// TIA Portal V19 export
FUNCTION "JB_CALL" : Void   // FC127, LAD
TITLE = JUNCTION BENCH WELDER CALL
// stored: SetENOAutomatically false
BEGIN

REGION Network 1: Data In - Welder speed potentiometer
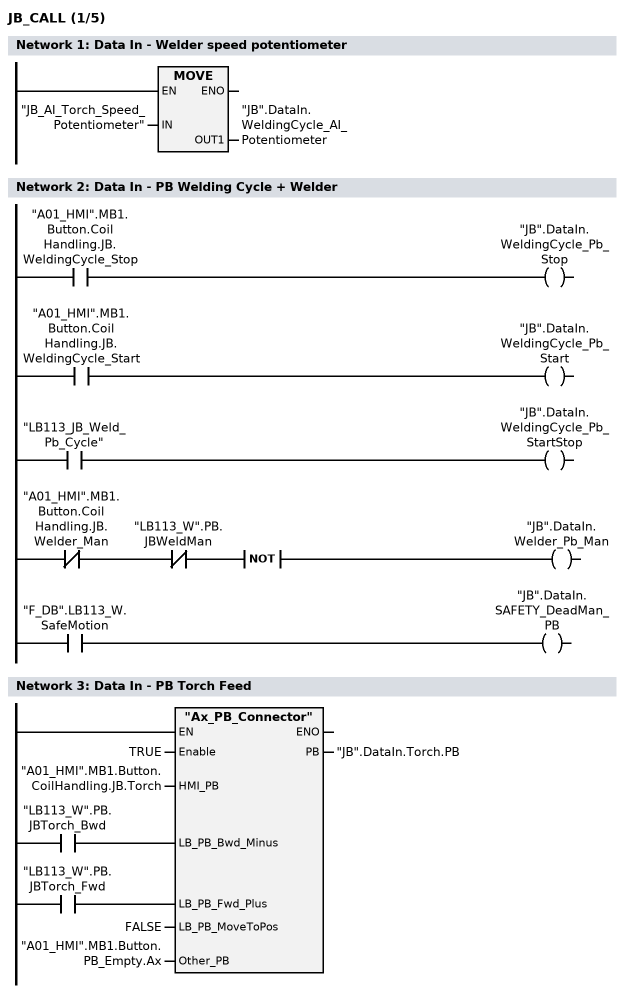
   RUNG wire#powerrail
      Move(in := "JB_AI_Torch_Speed_Potentiometer", out1 => "JB".DataIn.WeldingCycle_AI_Potentiometer)
   END_RUNG
   // the same network as SCL:
   "JB".DataIn.WeldingCycle_AI_Potentiometer := "JB_AI_Torch_Speed_Potentiometer";
END_REGION

REGION Network 2: Data In - PB Welding Cycle + Welder
   RUNG wire#powerrail
      Contact( "A01_HMI".MB1.Button.CoilHandling.JB.WeldingCycle_Stop )
      Coil( "JB".DataIn.WeldingCycle_Pb_Stop )
   END_RUNG
   RUNG wire#powerrail
      Contact( "A01_HMI".MB1.Button.CoilHandling.JB.WeldingCycle_Start )
      Coil( "JB".DataIn.WeldingCycle_Pb_Start )
   END_RUNG
   RUNG wire#powerrail
      Contact( "LB113_JB_Weld_Pb_Cycle" )
      Coil( "JB".DataIn.WeldingCycle_Pb_StartStop )
   END_RUNG
   RUNG wire#powerrail
      I_Contact( "A01_HMI".MB1.Button.CoilHandling.JB.Welder_Man )
      I_Contact( "LB113_W".PB.JBWeldMan )
      Not()
      Coil( "JB".DataIn.Welder_Pb_Man )
   END_RUNG
   RUNG wire#powerrail
      Contact( "F_DB".LB113_W.SafeMotion )
      Coil( "JB".DataIn.SAFETY_DeadMan_PB )
   END_RUNG
   // the same network as SCL:
   "JB".DataIn.WeldingCycle_Pb_Stop := "A01_HMI".MB1.Button.CoilHandling.JB.WeldingCycle_Stop;
   "JB".DataIn.WeldingCycle_Pb_Start := "A01_HMI".MB1.Button.CoilHandling.JB.WeldingCycle_Start;
   "JB".DataIn.WeldingCycle_Pb_StartStop := "LB113_JB_Weld_Pb_Cycle";
   "JB".DataIn.Welder_Pb_Man := NOT (NOT "A01_HMI".MB1.Button.CoilHandling.JB.Welder_Man AND NOT "LB113_W".PB.JBWeldMan);
   "JB".DataIn.SAFETY_DeadMan_PB := "F_DB".LB113_W.SafeMotion;
END_REGION

REGION Network 3: Data In - PB Torch Feed
   RUNG wire#powerrail
      "Ax_PB_Connector"(LB_PB_Bwd_Minus := wire#w1, LB_PB_Fwd_Plus := wire#w2, Enable := TRUE, HMI_PB := "A01_HMI".MB1.Button.CoilHandling.JB.Torch, LB_PB_MoveToPos := FALSE, Other_PB := "A01_HMI".MB1.Button.PB_Empty.Ax, PB => "JB".DataIn.Torch.PB)
   END_RUNG
   RUNG wire#powerrail
      Contact( "LB113_W".PB.JBTorch_Bwd )
   END_RUNG wire#w1
   RUNG wire#powerrail
      Contact( "LB113_W".PB.JBTorch_Fwd )
   END_RUNG wire#w2
   // the same network as SCL:
   "Ax_PB_Connector"(Enable := TRUE,
                     HMI_PB := "A01_HMI".MB1.Button.CoilHandling.JB.Torch,
                     LB_PB_Bwd_Minus := "LB113_W".PB.JBTorch_Bwd,
                     LB_PB_Fwd_Plus := "LB113_W".PB.JBTorch_Fwd,
                     LB_PB_MoveToPos := FALSE,
                     Other_PB := "A01_HMI".MB1.Button.PB_Empty.Ax,
                     PB => "JB".DataIn.Torch.PB);
END_REGION

REGION Network 4: Data In - PB Clamps
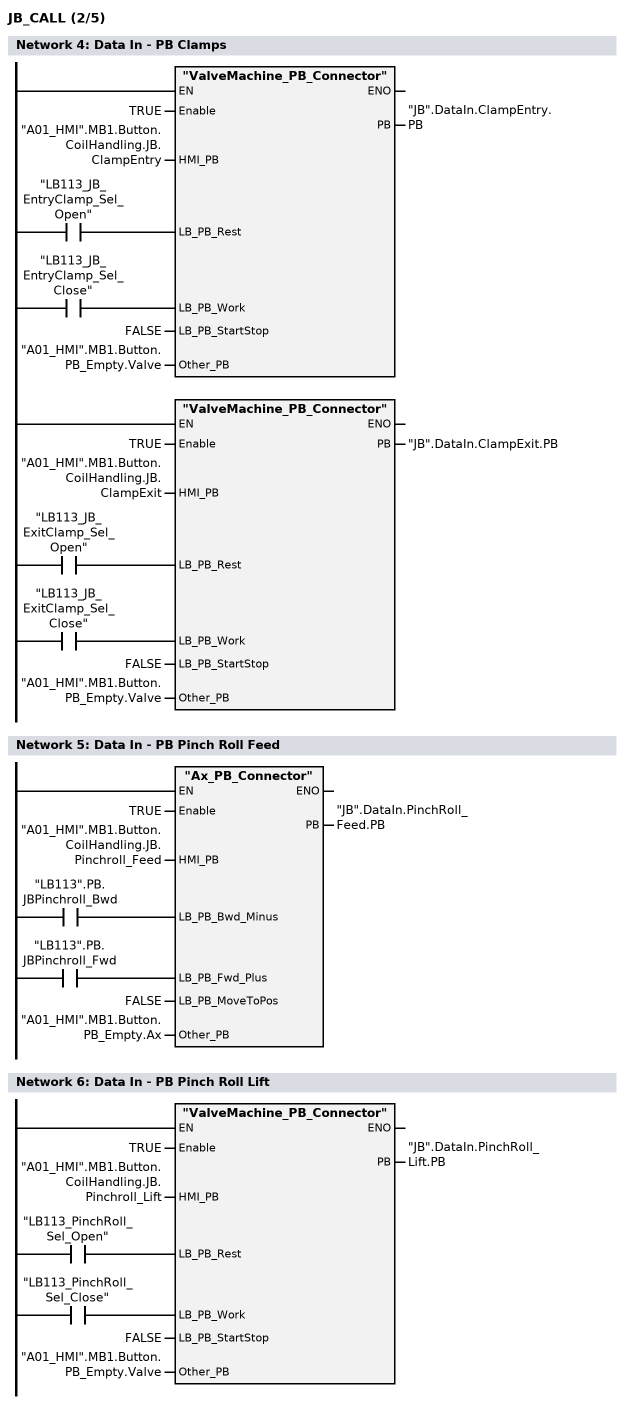
   RUNG wire#powerrail
      "ValveMachine_PB_Connector"(LB_PB_Rest := wire#w1, LB_PB_Work := wire#w2, Enable := TRUE, HMI_PB := "A01_HMI".MB1.Button.CoilHandling.JB.ClampEntry, LB_PB_StartStop := FALSE, Other_PB := "A01_HMI".MB1.Button.PB_Empty.Valve, PB => "JB".DataIn.ClampEntry.PB)
   END_RUNG
   RUNG wire#powerrail
      Contact( "LB113_JB_EntryClamp_Sel_Open" )
   END_RUNG wire#w1
   RUNG wire#powerrail
      Contact( "LB113_JB_EntryClamp_Sel_Close" )
   END_RUNG wire#w2
   RUNG wire#powerrail
      "ValveMachine_PB_Connector"(LB_PB_Rest := wire#w3, LB_PB_Work := wire#w4, Enable := TRUE, HMI_PB := "A01_HMI".MB1.Button.CoilHandling.JB.ClampExit, LB_PB_StartStop := FALSE, Other_PB := "A01_HMI".MB1.Button.PB_Empty.Valve, PB => "JB".DataIn.ClampExit.PB)
   END_RUNG
   RUNG wire#powerrail
      Contact( "LB113_JB_ExitClamp_Sel_Open" )
   END_RUNG wire#w3
   RUNG wire#powerrail
      Contact( "LB113_JB_ExitClamp_Sel_Close" )
   END_RUNG wire#w4
   // the same network as SCL:
   "ValveMachine_PB_Connector"(Enable := TRUE,
                           HMI_PB := "A01_HMI".MB1.Button.CoilHandling.JB.ClampEntry,
                           LB_PB_Rest := "LB113_JB_EntryClamp_Sel_Open",
                           LB_PB_Work := "LB113_JB_EntryClamp_Sel_Close",
                           LB_PB_StartStop := FALSE,
                           Other_PB := "A01_HMI".MB1.Button.PB_Empty.Valve,
                           PB => "JB".DataIn.ClampEntry.PB);
   "ValveMachine_PB_Connector"(Enable := TRUE,
                           HMI_PB := "A01_HMI".MB1.Button.CoilHandling.JB.ClampExit,
                           LB_PB_Rest := "LB113_JB_ExitClamp_Sel_Open",
                           LB_PB_Work := "LB113_JB_ExitClamp_Sel_Close",
                           LB_PB_StartStop := FALSE,
                           Other_PB := "A01_HMI".MB1.Button.PB_Empty.Valve,
                           PB => "JB".DataIn.ClampExit.PB);
END_REGION

REGION Network 5: Data In - PB Pinch Roll Feed
   RUNG wire#powerrail
      "Ax_PB_Connector"(LB_PB_Bwd_Minus := wire#w1, LB_PB_Fwd_Plus := wire#w2, Enable := TRUE, HMI_PB := "A01_HMI".MB1.Button.CoilHandling.JB.Pinchroll_Feed, LB_PB_MoveToPos := FALSE, Other_PB := "A01_HMI".MB1.Button.PB_Empty.Ax, PB => "JB".DataIn.PinchRoll_Feed.PB)
   END_RUNG
   RUNG wire#powerrail
      Contact( "LB113".PB.JBPinchroll_Bwd )
   END_RUNG wire#w1
   RUNG wire#powerrail
      Contact( "LB113".PB.JBPinchroll_Fwd )
   END_RUNG wire#w2
   // the same network as SCL:
   "Ax_PB_Connector"(Enable := TRUE,
                     HMI_PB := "A01_HMI".MB1.Button.CoilHandling.JB.Pinchroll_Feed,
                     LB_PB_Bwd_Minus := "LB113".PB.JBPinchroll_Bwd,
                     LB_PB_Fwd_Plus := "LB113".PB.JBPinchroll_Fwd,
                     LB_PB_MoveToPos := FALSE,
                     Other_PB := "A01_HMI".MB1.Button.PB_Empty.Ax,
                     PB => "JB".DataIn.PinchRoll_Feed.PB);
END_REGION

REGION Network 6: Data In - PB Pinch Roll Lift
   RUNG wire#powerrail
      "ValveMachine_PB_Connector"(LB_PB_Rest := wire#w1, LB_PB_Work := wire#w2, Enable := TRUE, HMI_PB := "A01_HMI".MB1.Button.CoilHandling.JB.Pinchroll_Lift, LB_PB_StartStop := FALSE, Other_PB := "A01_HMI".MB1.Button.PB_Empty.Valve, PB => "JB".DataIn.PinchRoll_Lift.PB)
   END_RUNG
   RUNG wire#powerrail
      Contact( "LB113_PinchRoll_Sel_Open" )
   END_RUNG wire#w1
   RUNG wire#powerrail
      Contact( "LB113_PinchRoll_Sel_Close" )
   END_RUNG wire#w2
   // the same network as SCL:
   "ValveMachine_PB_Connector"(Enable := TRUE,
                           HMI_PB := "A01_HMI".MB1.Button.CoilHandling.JB.Pinchroll_Lift,
                           LB_PB_Rest := "LB113_PinchRoll_Sel_Open",
                           LB_PB_Work := "LB113_PinchRoll_Sel_Close",
                           LB_PB_StartStop := FALSE,
                           Other_PB := "A01_HMI".MB1.Button.PB_Empty.Valve,
                           PB => "JB".DataIn.PinchRoll_Lift.PB);
END_REGION

REGION Network 7: Data In - PB Cut Head
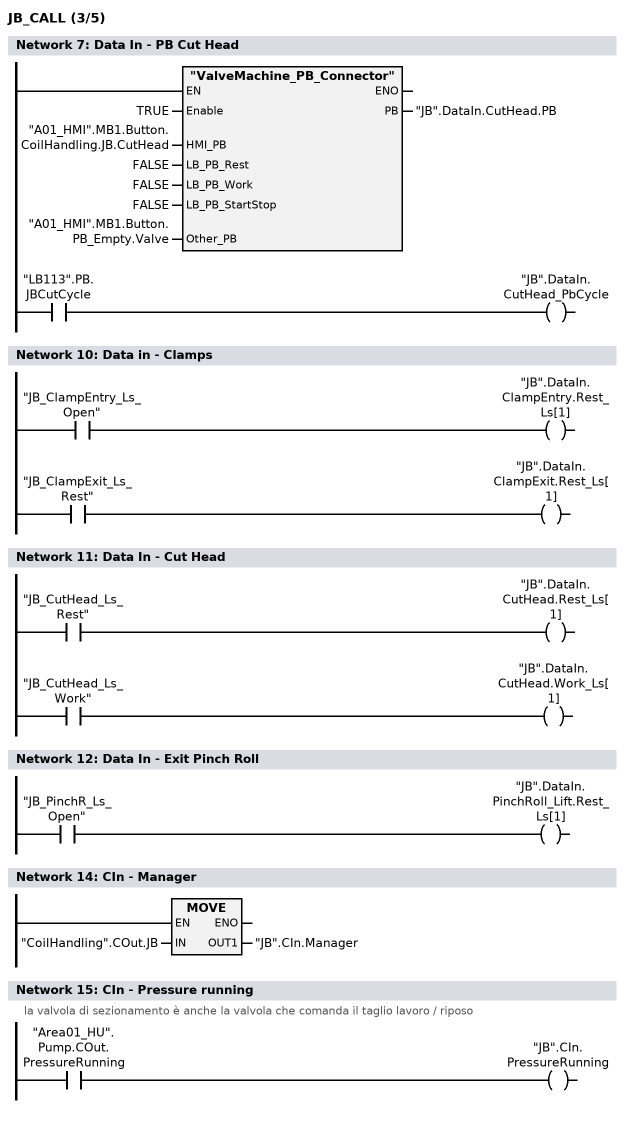
   RUNG wire#powerrail
      "ValveMachine_PB_Connector"(Enable := TRUE, HMI_PB := "A01_HMI".MB1.Button.CoilHandling.JB.CutHead, LB_PB_Rest := FALSE, LB_PB_Work := FALSE, LB_PB_StartStop := FALSE, Other_PB := "A01_HMI".MB1.Button.PB_Empty.Valve, PB => "JB".DataIn.CutHead.PB)
   END_RUNG
   RUNG wire#powerrail
      Contact( "LB113".PB.JBCutCycle )
      Coil( "JB".DataIn.CutHead_PbCycle )
   END_RUNG
   // the same network as SCL:
   "ValveMachine_PB_Connector"(Enable := TRUE,
                           HMI_PB := "A01_HMI".MB1.Button.CoilHandling.JB.CutHead,
                           LB_PB_Rest := FALSE,
                           LB_PB_Work := FALSE,
                           LB_PB_StartStop := FALSE,
                           Other_PB := "A01_HMI".MB1.Button.PB_Empty.Valve,
                           PB => "JB".DataIn.CutHead.PB);
   "JB".DataIn.CutHead_PbCycle := "LB113".PB.JBCutCycle;
END_REGION

REGION Network 8: >
END_REGION

REGION Network 9: >
END_REGION

REGION Network 10: Data in - Clamps
   RUNG wire#powerrail
      Contact( "JB_ClampEntry_Ls_Open" )
      Coil( "JB".DataIn.ClampEntry.Rest_Ls[1] )
   END_RUNG
   RUNG wire#powerrail
      Contact( "JB_ClampExit_Ls_Rest" )
      Coil( "JB".DataIn.ClampExit.Rest_Ls[1] )
   END_RUNG
   // the same network as SCL:
   "JB".DataIn.ClampEntry.Rest_Ls[1] := "JB_ClampEntry_Ls_Open";
   "JB".DataIn.ClampExit.Rest_Ls[1] := "JB_ClampExit_Ls_Rest";
END_REGION

REGION Network 11: Data In - Cut Head
   RUNG wire#powerrail
      Contact( "JB_CutHead_Ls_Rest" )
      Coil( "JB".DataIn.CutHead.Rest_Ls[1] )
   END_RUNG
   RUNG wire#powerrail
      Contact( "JB_CutHead_Ls_Work" )
      Coil( "JB".DataIn.CutHead.Work_Ls[1] )
   END_RUNG
   // the same network as SCL:
   "JB".DataIn.CutHead.Rest_Ls[1] := "JB_CutHead_Ls_Rest";
   "JB".DataIn.CutHead.Work_Ls[1] := "JB_CutHead_Ls_Work";
END_REGION

REGION Network 12: Data In - Exit Pinch Roll
   RUNG wire#powerrail
      Contact( "JB_PinchR_Ls_Open" )
      Coil( "JB".DataIn.PinchRoll_Lift.Rest_Ls[1] )
   END_RUNG
   // the same network as SCL:
   "JB".DataIn.PinchRoll_Lift.Rest_Ls[1] := "JB_PinchR_Ls_Open";
END_REGION

REGION Network 13: >
END_REGION

REGION Network 14: CIn - Manager
   RUNG wire#powerrail
      Move(in := "CoilHandling".COut.JB, out1 => "JB".CIn.Manager)
   END_RUNG
   // the same network as SCL:
   "JB".CIn.Manager := "CoilHandling".COut.JB;
END_REGION

REGION Network 15: CIn - Pressure running
   // la valvola di sezionamento è anche la valvola che comanda il taglio lavoro / riposo
   RUNG wire#powerrail
      Contact( "Area01_HU".Pump.COut.PressureRunning )
      Coil( "JB".CIn.PressureRunning )
   END_RUNG
   // the same network as SCL:
   "JB".CIn.PressureRunning := "Area01_HU".Pump.COut.PressureRunning;
END_REGION

REGION Network 16: >
END_REGION

REGION Network 17 (SCL): DSI
   "JB".DSI.Torch := "F_DB".DSI_S120_JB_Torch;

   "JB".DSI.PinchRoll_Feed := "F_DB".DSI_S120_JB_PinchRoll;

   "JB".DSI.ClampEntry :=
   "JB".DSI.ClampExit :=
   "JB".DSI.PinchRoll_Lift := "F_DB".DSI_V_Air_Gen;


   // Cut Head
   IF "JB".CutHead.COut.Rest_CheckNext THEN

       "JB".DSI.CutHead.SafeStop := "F_DB".DSI_V_JB_Cut_Rest.SafeStop;
       "JB".DSI.CutHead.PowerEnable := "F_DB".DSI_V_JB_Cut_Rest.PowerEnable;
       "JB".DSI.CutHead.DevicesInSafeState := "F_DB".DSI_V_JB_Cut_Rest.DevicesInSafeState;

   ELSIF "JB".CutHead.COut.Work_CheckNext THEN

       "JB".DSI.CutHead.SafeStop := "F_DB".DSI_V_JB_Cut_Work.SafeStop;
       "JB".DSI.CutHead.PowerEnable := "F_DB".DSI_V_JB_Cut_Work.PowerEnable;
       "JB".DSI.CutHead.DevicesInSafeState := "F_DB".DSI_V_JB_Cut_Work.DevicesInSafeState;

   ELSE
       "JB".DSI.CutHead.SafeStop := TRUE;
       "JB".DSI.CutHead.PowerEnable := FALSE;
       "JB".DSI.CutHead.DevicesInSafeState := TRUE;
   END_IF;
END_REGION

REGION Network 18 (SCL): Drive
   "JB".Drive.Torch.Infeed_ON := "Areas_ITF".AG.Infeed_Running;
   "JB".Drive.Torch.AccessPoint := "HW_Const_Values".CU1_PN_890A1_1_ModuleAccessPoint;
   "JB".Drive.Torch.AxisID := "CU1_ID_7_890A1_1_890M1";
   "JB".Drive.Torch.TokenChain := "TOKENCHAIN_CU1";

   "JB".Drive.Picnhroll_Feed.Infeed_ON := "Areas_ITF".AG.Infeed_Running;
   "JB".Drive.Picnhroll_Feed.AccessPoint := "CU1~PN~890A1_2_ModuleAccessPoint";
   "JB".Drive.Picnhroll_Feed.AxisID := "CU1_ID_8_890A1_2_900M1";
   "JB".Drive.Picnhroll_Feed.TokenChain := "TOKENCHAIN_CU1";
END_REGION

REGION Network 19 (SCL): HW ID
   "JB".HWID.Torch_TEL1 := "HW_Const_Values".CU1_PN_890A1_1_Standard_telegram_1;
   "JB".HWID.Pinchroll_Feed_TEL1 := "HW_Const_Values".CU1_PN_890A1_2_Standard_telegram_1;
   "JB".HWID.TorchEnc_IO := "HW_Const_Values".HW_894P1_Telegram_81_DI_DO;
END_REGION

REGION Network 20: >
END_REGION

REGION Network 21: Machine Manager
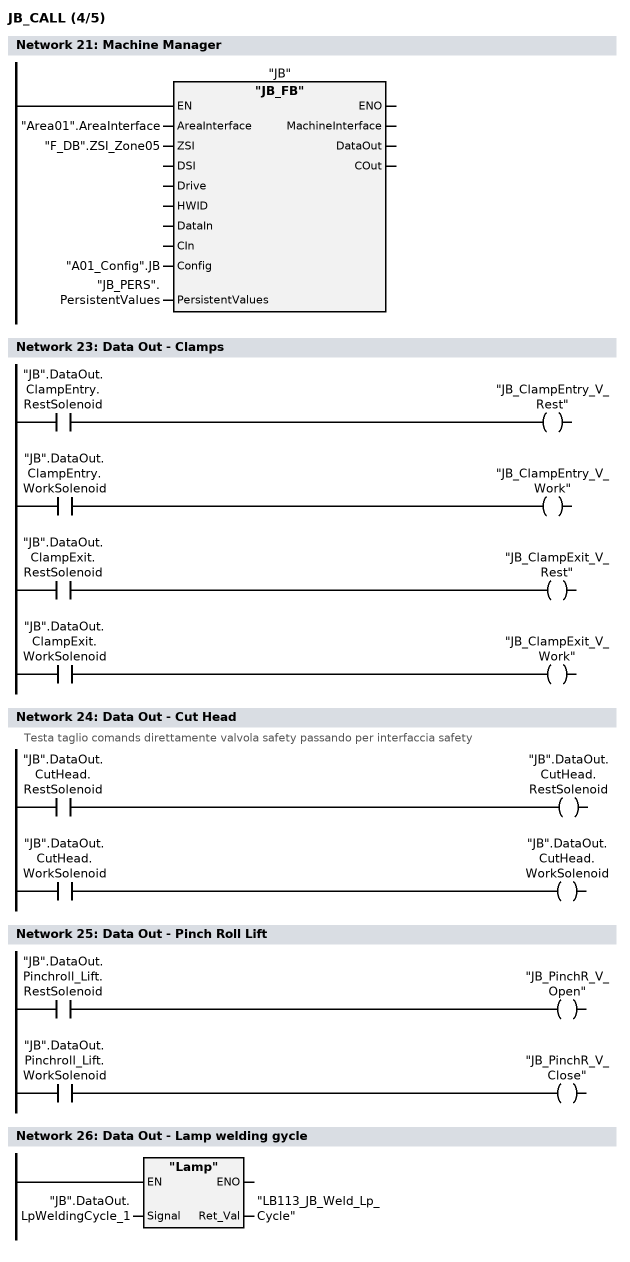
   RUNG wire#powerrail
      "JB"(AreaInterface := "Area01".AreaInterface, ZSI := "F_DB".ZSI_Zone05, DSI :=, Drive :=, HWID :=, DataIn :=, CIn :=, Config := "A01_Config".JB, PersistentValues := "JB_PERS".PersistentValues, MachineInterface =>, DataOut =>, COut =>)
   END_RUNG
   // the same network as SCL:
   "JB"(AreaInterface := "Area01".AreaInterface,   // "JB_FB"
        ZSI := "F_DB".ZSI_Zone05,
        Config := "A01_Config".JB,
        PersistentValues := "JB_PERS".PersistentValues);
END_REGION

REGION Network 22: >
END_REGION

REGION Network 23: Data Out - Clamps
   RUNG wire#powerrail
      Contact( "JB".DataOut.ClampEntry.RestSolenoid )
      Coil( "JB_ClampEntry_V_Rest" )
   END_RUNG
   RUNG wire#powerrail
      Contact( "JB".DataOut.ClampEntry.WorkSolenoid )
      Coil( "JB_ClampEntry_V_Work" )
   END_RUNG
   RUNG wire#powerrail
      Contact( "JB".DataOut.ClampExit.RestSolenoid )
      Coil( "JB_ClampExit_V_Rest" )
   END_RUNG
   RUNG wire#powerrail
      Contact( "JB".DataOut.ClampExit.WorkSolenoid )
      Coil( "JB_ClampExit_V_Work" )
   END_RUNG
   // the same network as SCL:
   "JB_ClampEntry_V_Rest" := "JB".DataOut.ClampEntry.RestSolenoid;
   "JB_ClampEntry_V_Work" := "JB".DataOut.ClampEntry.WorkSolenoid;
   "JB_ClampExit_V_Rest" := "JB".DataOut.ClampExit.RestSolenoid;
   "JB_ClampExit_V_Work" := "JB".DataOut.ClampExit.WorkSolenoid;
END_REGION

REGION Network 24: Data Out - Cut Head
   // Testa taglio comands direttamente valvola safety passando per interfaccia safety
   RUNG wire#powerrail
      Contact( "JB".DataOut.CutHead.RestSolenoid )
      Coil( "JB".DataOut.CutHead.RestSolenoid )
   END_RUNG
   RUNG wire#powerrail
      Contact( "JB".DataOut.CutHead.WorkSolenoid )
      Coil( "JB".DataOut.CutHead.WorkSolenoid )
   END_RUNG
   // the same network as SCL:
   "JB".DataOut.CutHead.RestSolenoid := "JB".DataOut.CutHead.RestSolenoid;
   "JB".DataOut.CutHead.WorkSolenoid := "JB".DataOut.CutHead.WorkSolenoid;
END_REGION

REGION Network 25: Data Out - Pinch Roll Lift
   RUNG wire#powerrail
      Contact( "JB".DataOut.Pinchroll_Lift.RestSolenoid )
      Coil( "JB_PinchR_V_Open" )
   END_RUNG
   RUNG wire#powerrail
      Contact( "JB".DataOut.Pinchroll_Lift.WorkSolenoid )
      Coil( "JB_PinchR_V_Close" )
   END_RUNG
   // the same network as SCL:
   "JB_PinchR_V_Open" := "JB".DataOut.Pinchroll_Lift.RestSolenoid;
   "JB_PinchR_V_Close" := "JB".DataOut.Pinchroll_Lift.WorkSolenoid;
END_REGION

REGION Network 26: Data Out - Lamp welding gycle
   RUNG wire#powerrail
      "Lamp"(Signal := "JB".DataOut.LpWeldingCycle_1, Ret_Val => "LB113_JB_Weld_Lp_Cycle")
   END_RUNG
   // the same network as SCL:
   "LB113_JB_Weld_Lp_Cycle" := "Lamp"(Signal := "JB".DataOut.LpWeldingCycle_1);
END_REGION

REGION Network 27: Data Out - Welder interface signal (START)
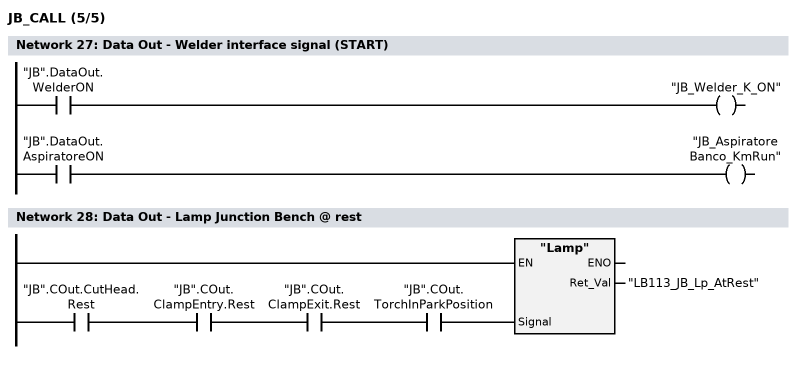
   RUNG wire#powerrail
      Contact( "JB".DataOut.WelderON )
      Coil( "JB_Welder_K_ON" )
   END_RUNG
   RUNG wire#powerrail
      Contact( "JB".DataOut.AspiratoreON )
      Coil( "JB_AspiratoreBanco_KmRun" )
   END_RUNG
   // the same network as SCL:
   "JB_Welder_K_ON" := "JB".DataOut.WelderON;
   "JB_AspiratoreBanco_KmRun" := "JB".DataOut.AspiratoreON;
END_REGION

REGION Network 28: Data Out - Lamp Junction Bench @ rest
   RUNG wire#powerrail
      "Lamp"(Signal := wire#w1, Ret_Val => "LB113_JB_Lp_AtRest")
   END_RUNG
   RUNG wire#powerrail
      Contact( "JB".COut.CutHead.Rest )
      Contact( "JB".COut.ClampEntry.Rest )
      Contact( "JB".COut.ClampExit.Rest )
      Contact( "JB".COut.TorchInParkPosition )
   END_RUNG wire#w1
   // the same network as SCL:
   "LB113_JB_Lp_AtRest" := "Lamp"(Signal := "JB".COut.CutHead.Rest AND "JB".COut.ClampEntry.Rest AND "JB".COut.ClampExit.Rest AND "JB".COut.TorchInParkPosition);
END_REGION
END_FUNCTION
